FUNCTION_BLOCK FB_ProtectRelay_SepamS48 EXTENDS FB_ProtectRelay_Base
//////////////////
// SEPAM system for High Voltage or Low Voltage Grid Protection. 
//////////////////

VAR_INPUT PERSISTENT
	// Parameters of the Object (instance/model specific) 
	   ParamTimeoutRTU						: TIME  := T#10S;					(* (s)	  Com RTU Timeout *)
	   ParamUnitID							: BYTE 	:= 1;						(* (NA)	  unit ID*)
	   ParamInInterfaceSub					: BOOL;								(* (NA)   Serial interface RS422/RS485 TYPE (0:EL6021, 1:SUB9)*)
END_VAR

VAR_OUTPUT		
                                 			                                                        
	OUT_UminLong							: BOOL; 							(* (NA) Long GTE fault or 3x Short GTE*)
	
END_VAR

VAR_INPUT
	// I/O Inputs	
	IN_MesAlarmIMax_IO						: BOOL; 							// I max fault Fault, Losing autorisation and not possible to consumed
	IN_MesAlarmUmin_IO						: BOOL; 							// U min Fault, Keeping autorisation, If we have 3 gte in 30 min ==> Stop fedding and consumed during 2h
	IN_MesAlarmPWH_IO						: BOOL; 							// Defaut wattmétrique
	                                                								                                                	
	IN_CmdReset_3GTEFault					: BOOL; 							// 3GTE Fault Reset 
	MesDataExd						 		: ProtectRelay_S48; 
	   	
END_VAR

VAR
	//M_Read
	Trig_Read								: R_TRIG;
	ModbusRTU								: FB_ModbusRTU ;					// (NA) FB for Modbus Reading
	MbStruct								: ARRAY[1..2] OF Struct_InputRTU;

                                			
	ModbusAlarm								: ARRAY[1..2] OF BOOL;				// (NA) Read alarm
	AX_Quantity								: ARRAY[1..2] OF WORD;				// (NA) Quantity of blocks to read
	AX_Address								: ARRAY[1..2] OF WORD;				// (NA) Start address of the read
	OutErrorMbRead							: ARRAY[1..2] OF BOOL;
                                			
	Busy									: BOOL;
	MesBlock_Temp							: ARRAY [1..2] OF ARRAY [0..94] OF WORD;
	                            			
	RTrigI									: R_TRIG;
                         			
	//M_EVALUATE                			
	TON_GteIsLong							: TON;

	FB_3GTE									: FB_CountNinTimeWindow; 
	
	R_TRIG_GTE3Time							: R_TRIG;

END_VAR

METHOD M_AlarmManagement
//////////////////
// Manages Sepam Alarms. Alarms opens HT CB until Sepam manual reset. Warning opens CB-L but does not maintain warning.
/////////////////

VAR 
	// Method local variables (reinitialized at each cycle) 
	FB_AlarmCodeManager 	: FB_AlarmCodeManager ; 
 	ComWarning				: BOOL;
	ComAlarms				: BOOL;
END_VAR
ComWarning	:= OutErrorMbRead[1] OR OutErrorMbRead[2];
ComAlarms	:= OutErrorMbRead[1];

TON_ComAlarm(IN:= ComAlarms , PT:= ParamTempoComAlarm, Q=> MesDataExd.MesData.MesAlarmCom) ;	

// ALARM CODE //
	FB_AlarmCodeManager(
		bAlarm1				:= MesDataExd.MesData.MesAlarmUmin , 		// Min U Fault 
		bAlarm2				:= FALSE ,									//
		bAlarm3				:= NOT IN_MesWatchDog_IO,					// Watchdog TRUE := OK, False = Dead #COM
		bAlarm4				:= MesDataExd.MesData.MesAlarmImax,     	// C13100 Fault (Max I) 
		bAlarm5				:= FALSE,         							// 
		bAlarm6				:= FALSE, 									// 
		bAlarm7				:= FALSE, 									// 
		bAlarm8				:= FALSE, 									// 
		bAlarm9				:= FALSE, 									// 
		bAlarm10			:= FALSE, 									// 
		bAlarm11			:= FALSE, 									// 
		bAlarm12			:= FALSE, 									// 
		bAlarm13			:= FALSE, 									// 
		bAlarm14			:= FALSE, 									// 
		bAlarm15			:= FALSE ,									//  	
		wAlarmCode			=>MesDataExd.MesData.MesAlarmCode);

// WARNING CODE //
	FB_AlarmCodeManager(
		bAlarm1			:= ComWarning, 									// At least one register do not respond #COM
		bAlarm2			:= MesDataExd.MesData.MesAlarmCom ,				// Communication alarm #COM
		bAlarm3			:= FALSE , 										//		
		bAlarm4			:= FALSE , 										//
		bAlarm5			:= FALSE , 										//
		bAlarm6			:= IN_MesAlarmPWH_IO, 							// Wattmetric fault	
		bAlarm7			:= MesDataExd.MesData.MesAlarmUmin_Long, 		// Long Min U Fault (> 50s)
		bAlarm8			:= MesDataExd.MesData.MesAlarm_GTE3Time, 		// 3 min U fault in a row (GTE 3 times)
		bAlarm9			:= FALSE, 										//
		bAlarm10		:= FALSE, 										//
		bAlarm11		:= FALSE, 										//
		bAlarm12		:= FALSE, 										//
		bAlarm13		:= FALSE, 										//
		bAlarm14		:= FALSE, 										//
		bAlarm15		:= FALSE, 										//
		wAlarmCode		=>MesDataExd.MesData.MesWarningCode);

// EVENT CODE //
	FB_AlarmCodeManager(
		bAlarm1			:=FALSE, 										// 
		bAlarm2			:=FALSE, 										// 
		bAlarm3			:=FALSE, 										// 
		bAlarm4			:=FALSE, 										// 
		bAlarm5			:=FALSE, 										//
		bAlarm6			:=FALSE, 										//
		bAlarm7			:=FALSE, 										//
		bAlarm8			:=FALSE, 										//
		bAlarm9			:=FALSE, 										//
		bAlarm10		:=FALSE, 										//
		bAlarm11		:=FALSE, 										//
		bAlarm12		:=FALSE, 										//
		bAlarm13		:=FALSE, 										//
		bAlarm14		:=FALSE, 										//
		bAlarm15		:=FALSE, 										//
		wAlarmCode		=>MesDataExd.MesData.MesEventCode);
END_METHOD

METHOD M_CP 
VAR_INPUT
END_VAR


SUPER^.M_CP() ; 




Trig_Cmd_Read(CLK:=IN_CmdToggleRead);
Trig_Cmd_Write(CLK:=IN_CmdToggleWrite);
	
IF Trig_Cmd_Read.Q THEN
	IN_CmdToggleRead := FALSE;
	MesDataExd.MesData.MesCP_Read := NOT MesDataExd.MesData.MesCP_Read;
END_IF


IF Trig_Cmd_Write.Q THEN
	IN_CmdToggleWrite := FALSE;
	MesDataExd.MesData.MesCP_Write := NOT MesDataExd.MesData.MesCP_Write;
END_IF
END_METHOD

METHOD M_Evaluate
VAR_INPUT
END_VAR

VAR

END_VAR
// GTE IS LONG AFTER 50S

TON_GteIsLong(IN:=IN_MesAlarmUmin_IO ,PT:=T#50S); 

FB_3GTE(IN_bInput := IN_MesAlarmUmin_IO , IN_bReset := IN_CmdReset_3GTEFault , IN_CountMax := 3 , ParamTimeToMeasure := T#30M , OUT_FlagNinT =>MesDataExd.MesData.MesAlarm_GTE3Time ) ; 
	
MesDataExd.MesData.MesAlarmUmin_Long := TON_GteIsLong.Q; 


//Update MesData
MesDataExd.MesData.MesI			:= (MesDataExd.MesData.MesI1 + MesDataExd.MesData.MesI2 + MesDataExd.MesData.MesI3) / 3 ;
MesDataExd.MesData.MesAlarmUmin := IN_MesAlarmUmin_IO;
MesDataExd.MesData.MesAlarmImax	:= IN_MesAlarmIMax_IO;

R_TRIG_GTE3Time (CLK := A1_SUBMV.A1_ProtectRelay.MesDataExd.MesData.MesAlarm_GTE3Time);

OUT_UminLong := A1_SUBMV.A1_ProtectRelay.MesDataExd.MesData.MesAlarmUmin_Long OR R_TRIG_GTE3Time.Q;
END_METHOD

METHOD M_Init
VAR_INPUT
END_VAR
END_METHOD

METHOD M_Read
//////////////////
//  Method Calls 
/////////////////

VAR 
	MW 					: FB_MergeWordsToDint; 
	KK : UINT;

	AX_Addr					: ARRAY[1..2] OF UINT 	:= [16#113,		16#10B];
	AX_Qty					: ARRAY[1..2] OF UINT	:= [94,			1];
	AX_UnitId				: ARRAY[1..2] OF BYTE	:= [1,			1];
	AX_Function				: ARRAY[1..2] OF UINT	:= [3,			3];	
	AX_Priority				: ARRAY[1..2] OF UINT	:= [1,			1];
END_VAR
// CP-Read / Write 


IF MesDataExd.MesData.MesCP_Read  THEN	
	
	
	ModbusRTU();
	Trig_Read(Clk := CalLocalTimeStruct.wMilliseconds < 200);
	IF Trig_Read.Q THEN
		FOR KK := 1 TO 2 DO
				ModbusRTU.M_AddAction_FIFO(InStruct := MbStruct[KK], InPriority := AX_Priority[KK]);
		END_FOR
	END_IF
	
	MbStruct[1].InBuffer 	:= ADR(MesBlock_Temp[1]);
	MbStruct[1].InFunction 	:= AX_Function[1];
	MbStruct[1].InQuantity 	:= AX_Qty[1];
	MbStruct[1].InStartAddr := AX_Addr[1];
	MbStruct[1].InUnitID 	:= AX_UnitId[1];
	
	MbStruct[2].InBuffer 	:= ADR(MesBlock_Temp[2]);
	MbStruct[2].InFunction 	:= AX_Function[2];
	MbStruct[2].InQuantity 	:= AX_Qty[2];
	MbStruct[2].InStartAddr := AX_Addr[2];
	MbStruct[2].InUnitID 	:= AX_UnitId[2];
	
	MW( WORD_STRONG:= MesBlock_Temp[1][0], SIGNED:=FALSE, FIX:=1 , SIZE:=1, VAR_OUT := MesDataExd.MesData.MesI1);
	MW( WORD_STRONG:= MesBlock_Temp[1][1], SIGNED:=FALSE, FIX:=1 , SIZE:=1, VAR_OUT := MesDataExd.MesData.MesI2);
	MW( WORD_STRONG:= MesBlock_Temp[1][2], SIGNED:=FALSE, FIX:=1 , SIZE:=1, VAR_OUT := MesDataExd.MesData.MesI3);
	MW( WORD_STRONG:= MesBlock_Temp[1][4], SIGNED:=FALSE, FIX:=1 , SIZE:=1, VAR_OUT := MesDataExd.MesData.MesI0);
	MW( WORD_STRONG:= MesBlock_Temp[1][8], SIGNED:=FALSE, FIX:=1 , SIZE:=1, VAR_OUT := MesDataExd.MesData.MesImax1);
	MW( WORD_STRONG:= MesBlock_Temp[1][9], SIGNED:=FALSE, FIX:=1 , SIZE:=1, VAR_OUT := MesDataExd.MesData.MesImax2);
	MW( WORD_STRONG:= MesBlock_Temp[1][10], SIGNED:=FALSE, FIX:=1 , SIZE:=1, VAR_OUT := MesDataExd.MesData.MesImax3);
	MW( WORD_STRONG:= MesBlock_Temp[1][14], SIGNED:=FALSE, FIX:=0 , SIZE:=1, VAR_OUT := MesDataExd.MesV1);
	MW( WORD_STRONG:= MesBlock_Temp[1][15], SIGNED:=FALSE, FIX:=0 , SIZE:=1, VAR_OUT := MesDataExd.MesV2);
	MW( WORD_STRONG:= MesBlock_Temp[1][16], SIGNED:=FALSE, FIX:=0 , SIZE:=1, VAR_OUT := MesDataExd.MesV3);
	MW( WORD_STRONG:= MesBlock_Temp[1][11], SIGNED:=FALSE, FIX:=0 , SIZE:=1, VAR_OUT := MesDataExd.MesData.MesU12);
	MW( WORD_STRONG:= MesBlock_Temp[1][12], SIGNED:=FALSE, FIX:=0 , SIZE:=1, VAR_OUT := MesDataExd.MesData.MesU31);
	MW( WORD_STRONG:= MesBlock_Temp[1][13], SIGNED:=FALSE, FIX:=0 , SIZE:=1, VAR_OUT := MesDataExd.MesData.MesU23);
	MW( WORD_STRONG:= MesBlock_Temp[1][20], SIGNED:=FALSE, FIX:=2 , SIZE:=1, VAR_OUT := MesDataExd.MesData.MesFreq);
	MW( WORD_STRONG:= MesBlock_Temp[1][21], SIGNED:=TRUE, FIX:=0 , SIZE:=1, VAR_OUT := MesDataExd.MesP);
	MW( WORD_STRONG:= MesBlock_Temp[1][22], SIGNED:=TRUE, FIX:=0 , SIZE:=1, VAR_OUT := MesDataExd.MesQ);
	MW( WORD_STRONG:= MesBlock_Temp[1][23], SIGNED:=TRUE, FIX:=0 , SIZE:=1, VAR_OUT := MesDataExd.MesS);
	MW( WORD_STRONG:= MesBlock_Temp[1][26], SIGNED:=TRUE, FIX:=2 , SIZE:=1, VAR_OUT := MesDataExd.MesCosPhi);
	MW( WORD_STRONG:= MesBlock_Temp[1][27], WORD_WEAK := MesBlock_Temp[1][28], SIGNED:=FALSE, FIX:=1 , SIZE:=2, VAR_OUT := MesDataExd.EActProd);
	MW( WORD_STRONG:= MesBlock_Temp[1][29], WORD_WEAK := MesBlock_Temp[1][30], SIGNED:=FALSE, FIX:=1 , SIZE:=2, VAR_OUT := MesDataExd.EActCons);
	MW( WORD_STRONG:= MesBlock_Temp[1][31], WORD_WEAK := MesBlock_Temp[1][32], SIGNED:=FALSE, FIX:=1 , SIZE:=2, VAR_OUT := MesDataExd.EReactProd);
	MW( WORD_STRONG:= MesBlock_Temp[1][33], WORD_WEAK := MesBlock_Temp[1][34], SIGNED:=FALSE, FIX:=1 , SIZE:=2, VAR_OUT := MesDataExd.EReactCons);
	
	
	MesDataExd.Input11 := MesBlock_Temp[2][0].0;
	MesDataExd.Input12 := MesBlock_Temp[2][0].1;
	MesDataExd.Input13 := MesBlock_Temp[2][0].2;
	MesDataExd.Input14 := MesBlock_Temp[2][0].3;
	MesDataExd.Input21 := MesBlock_Temp[2][0].4;
	MesDataExd.Input22 := MesBlock_Temp[2][0].5;
	MesDataExd.Input23 := MesBlock_Temp[2][0].6;
	MesDataExd.Input24 := MesBlock_Temp[2][0].7;
	MesDataExd.Input25 := MesBlock_Temp[2][0].8;
	MesDataExd.Input26 := MesBlock_Temp[2][0].9;

END_IF

// Properties Update 
	MesDataExd.MesU := (MesDataExd.MesData.MesU12 + MesDataExd.MesData.MesU31 + MesDataExd.MesData.MesU23 ) /3 ; 
	
	IF MesDataExd.MesP <> 0 THEN
		MesDataExd.MesTanPhi := MesDataExd.MesQ /MesDataExd.MesP;
	ELSE
		MesDataExd.MesTanPhi := 0;
	END_IF
END_METHOD

END_FUNCTION_BLOCK

(* stored: Version 1.1.0.1, ProductVersion 3.1.4024.12
   POU FB_ProtectRelay_SepamS48: Id {bc8eb8e4-4f1c-4671-84af-b4ab0a7ab1b7}, SpecialFunc None
   Method M_AlarmManagement: Id {7d768758-0d1b-46a4-8977-7d92b89c4fbc}
   Method M_CP: Id {620a8763-1206-454d-8242-2fc61a8b2a83}
   Method M_Evaluate: Id {ecb3d80c-3e98-496d-bb4f-107388ab39e6}
   Method M_Init: Id {00e284e9-24fa-406b-85ab-b9a977105e5b}
   Method M_Read: Id {f84e6537-fc67-4949-802f-02c126e24c2e} *)
